// TIA Portal V17 export
// export: Created 2025-03-05T08:02:05.3810133Z, ExportSetting WithDefaults, DisplayName Totally Integrated Automation Portal, DisplayVersion V17 Update 8, DisplayName TIA Portal Openness, DisplayVersion V17 Update 8, DisplayName TIA Portal Version Control Interface, DisplayVersion V17, DisplayName SINAMICS Startdrive Advanced, DisplayVersion V17 SP2, DisplayName SINAMICS Startdrive G110M, G120, G120C, G120D, G120P, G115D, DisplayVersion V17 SP2, DisplayName SINAMICS Startdrive G130, G150, S120, S150, SINAMICS MV, S210, DisplayVersion V17 SP2, DisplayName STEP 7 Professional, DisplayVersion V17 Update 8, DisplayName SINUMERIK ONE STEP 7 Toolbox, DisplayVersion V17 Update 12, DisplayName SINUMERIK 840D sl STEP 7 Toolbox, DisplayVersion V17 Update 12, DisplayName STEP 7 Safety, DisplayVersion V17 Update 6, DisplayName WinCC Advanced, DisplayVersion V17 Update 8
TYPE "LBP_typePowerrideOutput"
TITLE = Powerride image / Imagen de powerride / Powerride Abbild
// Output image of powerride / Imagen de salida de powerride / Ausgangsabbild von Powerride
// stored: IsFailsafeCompliant false
   STRUCT
      ledInfo : DWord;   // LED 24...LED 0 / Led24..Led0
      scaleRed : Bool;   // Wenn TRUE, leuchtet rotes LED-Band / when true, red scale LED is on / Si es TRUE, la franja de LED roja alumbra
      scaleGreen : Bool;   // Wenn TRUE, leuchtet grünes LED-Band / when true, green scale LED is on / Si es TRUE, la franja de LED verde alumbra
      scaleBlue : Bool;   // Wenn TRUE, leuchtet blaues LED-Band / when true, blue scale LED ist on / Si es TRUE, la franja de LED azul alumbra
      buttonRed : Bool;   // Wenn TRUE, leuchtet rote Taster-LED / when true, red push button LED is on / Si es TRUE, el pulsador LED rojo alumbra
      buttonGreen : Bool;   // Wenn TRUE, leuchtet grüne Taster-LED / when true, green push button LED is on / Si es TRUE, el pulsador LED verde alumbra
      buttonBlue : Bool;   // Wenn TRUE, leuchtet grüne Taster-LED / when true, green push button LED is on / Si es TRUE, el pulsador LED verde alumbra
      reserved46 : Bool;
      reserved47 : Bool;
      vibrationPattern : USInt;   // Zu verwendender Vibrationsmutserindex / vibration pattern index to be used / Índice de plantilla de vibración que ha de utilizarse
   END_STRUCT;
END_TYPE
